GVL_XTS.XtsTransport.GroupItf                   :=   GVL_XTS.CaGroupItf;
GVL_XTS.XtsTransport.GroupInfo                  REF= GVL_XTS.CaGroupInfo;
                                        
GVL_XTS.XtsTransport.MoverItf                   REF= GVL_XTS.MoverItf;
GVL_XTS.XtsTransport.MoverInfo                  REF= GVL_XTS.MoverInfo;
GVL_XTS.XtsTransport.MoverLastPosition          REF= GVL_XTS.LastPosition;
GVL_XTS.XtsTransport.MoverLastGap               REF= GVL_XTS.LastGap;

GVL_XTS.XtsTransport.StationStartIndex          :=   GVL_XTS.StationStartIndex;                                        
GVL_XTS.XtsTransport.StationStart               REF= GVL_XTS.StationStart;      // start position for E_XTS_TRANSPORT_CTRL.CMD_TRANSPORT_START
GVL_XTS.XtsTransport.StationCtrlItf             REF= GVL_XTS.StationCtrlItf;    // station interfaces are required for accessing station methods
GVL_XTS.XtsTransport.StationListsItf            REF= GVL_XTS.StationListItf;    // list interface is required for access to linked list methods
GVL_XTS.XtsTransport.StationControl             REF= GVL_XTS.StationCtrl;
GVL_XTS.XtsTransport.StationState               REF= GVL_XTS.StationState;
//############################################################################
// 	XTS Transport Unit/
//############################################################################
//############################################################################
//############################################################################
// 	/XTS Stations
//############################################################################	
FOR nStation := 1 TO MAX_STATION
DO
  // epimetheus assembles the body
  GVL_XTS.StationListItf[nStation]              := GVL_XTS.StationList[nStation];   // interfaces for list methods
  GVL_XTS.StationCtrlItf[nStation]              := GVL_XTS.Station[nStation];       // interfaces for station methods

  CASE GVL_XTS.StationParameter[nStation].eType
  OF
    //-----------------------------------------------------------------------------
    E_STATION_TYPE.STATION_PROCESS:
      GVL_XTS.Station[nStation].MessageLevel    := GVL_MSG_XTS.MessageLevelStations[nStation];

      GVL_XTS.Station[nStation].StationId       := nStation;  // Know Thyself!

    
      GVL_XTS.Station[nStation].Ctrl            REF= GVL_XTS.StationCtrl;           // station ctrl from extern
      GVL_XTS.Station[nStation].State           REF= GVL_XTS.StationState;          // station state to extern
    
      GVL_XTS.Station[nStation].ItfStations     REF= GVL_XTS.StationListItf;        // give every station all list interfaces for writing mover tickets
      GVL_XTS.Station[nStation].ItfMover        REF= GVL_XTS.MoverItf;              // give every station all mover interfaces for movement in / out of station
      GVL_XTS.Station[nStation].Mover           REF= GVL_XTS.AxisRefMover;          // AXIS_REF to read infos from
      GVL_XTS.Station[nStation].MoverOffset     REF= GVL_XTS.PositionOffset;        // static offsets for all stations, all movers, all stop positions
    
      GVL_XTS.Station[nStation].StationParameter  REF= GVL_XTS.StationParameter;// give every station all station parameters for sending to WaitPos of target station
    
      // cyclic call
      GVL_XTS.Station[nStation].Cycle();                                        // cycle for handshaking with extern
    
      // Queue data for each station
      GVL_XTS.StationQueue[nStation]            := GVL_XTS.StationListItf[nStation].Data;


    //-----------------------------------------------------------------------------
    E_STATION_TYPE.STATION_GEAR_IN_POS:
      GVL_XTS.StationGearIn[nStation].MessageLevel:= GVL_MSG_XTS.MessageLevelStations[nStation];

      GVL_XTS.StationGearIn[nStation].StationId   := nStation;  // Know Thyself!
    
      GVL_XTS.StationGearIn[nStation].Ctrl        REF= GVL_XTS.StationCtrl;           // station ctrl from extern
      GVL_XTS.StationGearIn[nStation].State       REF= GVL_XTS.StationState;          // station state to extern
    
      GVL_XTS.StationGearIn[nStation].ItfStations REF= GVL_XTS.StationListItf;        // give every station all list interfaces for writing mover tickets
      GVL_XTS.StationGearIn[nStation].ItfMover    REF= GVL_XTS.MoverItf;              // give every station all mover interfaces for movement in / out of station
      GVL_XTS.StationGearIn[nStation].Mover       REF= GVL_XTS.AxisRefMover;          // AXIS_REF to read infos from
      GVL_XTS.StationGearIn[nStation].MoverOffset REF= GVL_XTS.PositionOffset;        // static offsets for all stations, all movers, all stop positions
    
    
      GVL_XTS.StationGearIn[nStation].StationParameter  REF= GVL_XTS.StationParameter;// give every station all station parameters for sending to WaitPos of target station
    
      // cyclic call
      GVL_XTS.StationGearIn[nStation].Cycle();                                        // cycle for handshaking with extern
    
      // Queue data for each station
      GVL_XTS.StationQueue[nStation]            := GVL_XTS.StationListItf[nStation].Data;
  ELSE
      //---------------------------------------------------------------------------------
      // no valid station type --> no identity
      //---------------------------------------------------------------------------------
      GVL_XTS.Station[nStation].StationId       := 0; // I am no one
      //---------------------------------------------------------------------------------
  END_CASE
END_FOR
//############################################################################
// 	XTS Stations/
//############################################################################	
//############################################################################
//############################################################################
// 	/XPU environment
//############################################################################	
GVL_XTS.Xpu.XpuInstance                         :=   1;
GVL_XTS.Xpu.MessageLevel                        :=   GVL_MSG_XTS.MessageLevelXpu;

GVL_XTS.Xpu.Ctrl                                REF= GVL_XTS.XpuCtrl;
GVL_XTS.Xpu.State                               REF= GVL_XTS.XpuState;
GVL_XTS.Xpu.XpuModuleInfoData                   REF= GVL_XTS.XpuModules;

GVL_XTS.Xpu.CaGroupOID                          :=   GVL_XTS.CaGroup.GroupInfo.CaGroupOID;

// cyclic call                                
GVL_XTS.Xpu();                                
GVL_XTS.XpuInfo                                 :=   GVL_XTS.Xpu.XpuInfo;
//############################################################################
// 	XPU environment/
//############################################################################	
//############################################################################
//############################################################################	
// 	/CA-Group Class
//############################################################################
// message device identifier
GVL_XTS.CaGroup.MessageDeviceIndex              :=   e_Device.CaGroup + 1;	
// assignment
GVL_XTS.CaGroup.AxisRef                         REF= GVL_XTS.AxisRefMover;
// Interface to Mover methods
GVL_XTS.CaGroup.MoverItf                        REF= GVL_XTS.MoverItf; 
GVL_XTS.CaGroup.GroupRef                        REF= GVL_XTS.CaGroupRef;
GVL_XTS.CaGroup.XpuInfo                         REF= GVL_XTS.XpuInfo;
// cyclic call
GVL_XTS.CaGroup.InfoCycle(TRUE);                // read group status
// InfoData from group
GVL_XTS.CaGroupInfo                             :=   GVL_XTS.CaGroup.GroupInfo;
// Interface of CaGroup
GVL_XTS.CaGroupItf                              :=   GVL_XTS.CaGroup;
//############################################################################	
// 	CA-Group Class/
//############################################################################
//############################################################################
//############################################################################
//  /Mover Class	
//############################################################################	
FOR nMover := 1 TO MAX_MOVER
DO
  GVL_XTS.Mover[nMover].MoverId                 :=   nMover;
  GVL_XTS.Mover[nMover].RailLength              :=   GVL_XTS.Xpu.RailLength;  // mover needs RailLength, in order to calc absolute position from modulo input
  GVL_XTS.Mover[nMover].MessageLevel            :=   GVL_MSG_XTS.MessageLevelMovers[nMover];

  GVL_XTS.Mover[nMover].Ctrl                    REF= GVL_XTS.MoverCtrl;       // mover control from extern
  GVL_XTS.Mover[nMover].State                   REF= GVL_XTS.MoverState;      // mover state to extern

  GVL_XTS.Mover[nMover].MoveData                REF= GVL_XTS.MoveData;        // dyn constraints for extern to write
  GVL_XTS.Mover[nMover].GearData                REF= GVL_XTS.GearData;        // GearIn/GearInPosCa data fro extern to write

  // assignment
  GVL_XTS.Mover[nMover].Mover                   REF= GVL_XTS.AxisRefMover[nMover];  // axis reference to Mover function block
  GVL_XTS.Mover[nMover].LastGap                 REF= GVL_XTS.LastGap[nMover];       // reference to last used gap value datafield
  GVL_XTS.Mover[nMover].LastPosition            REF= GVL_XTS.LastPosition[nMover];  // reference to last position datafield

  GVL_XTS.Mover[nMover].MoverInfo		            REF= GVL_XTS.MoverInfo[nMover];     // refernence to mover info data (ActPos, SetPos, ...)

  GVL_XTS.MoverItf[nMover]                      :=   GVL_XTS.Mover[nMover];

  // cyclic call
  GVL_XTS.Mover[nMover].Cycle();                // call AXIS_REF()
  GVL_XTS.Mover[nMover]();                      // call Ctrl/State
END_FOR
//############################################################################
//  Mover Class/	
//############################################################################	
//############################################################################
//############################################################################
//  /Mover Selector	
//############################################################################
GVL_XTS.MoverSelector.Ctrl                      REF= GVL_XTS.MoverSelectorCtrl;
GVL_XTS.MoverSelector.State                     REF= GVL_XTS.MoverSelectorState;
GVL_XTS.MoverSelector.AxisRef                   REF= GVL_XTS.AxisRefMover;
GVL_XTS.MoverSelector.Info                      REF= GVL_XTS.MoverInfo;
GVL_XTS.MoverSelector.ItfMover                  REF= GVL_XTS.MoverItf;

GVL_XTS.MoverSelector();
//############################################################################
//  Mover Selector/	
//############################################################################	
//############################################################################
//############################################################################
//  /logging
//    - all life is problem solving
//############################################################################
GVL_MSG_XTS.TransportMessageData.Ctrl               REF= GVL_MSG_XTS.TransportMessageCtrl;
GVL_MSG_XTS.TransportMessageData.State              REF= GVL_MSG_XTS.TransportMessageState;
GVL_MSG_XTS.TransportMessageData.MessageIndex       REF= GVL_MSG_XTS.MessageTransportIndex;
GVL_MSG_XTS.TransportMessageData.ErrorIndex         REF= GVL_MSG_XTS.MessageTransportError;
GVL_MSG_XTS.TransportMessageData.DirRoot            :=   ADR(GVL_MSG_XTS.LOG_DIR);
GVL_MSG_XTS.TransportMessageData.FileRoot           :=   ADR(GVL_MSG_XTS.LOG_FILE);
GVL_MSG_XTS.TransportMessageData.MsgList            :=   ADR(GVL_MSG_XTS.TransportMessages);
GVL_MSG_XTS.TransportMessageData.LocalTime          :=   ADR(GVL_MSG_XTS.dtLocalTime);
GVL_MSG_XTS.TransportMessageData();
eMsgState                                       :=   f_GetState   (GVL_MSG_XTS.TransportMessageState.State);
eMsgProgress                                    :=   f_GetProgress(GVL_MSG_XTS.TransportMessageState.State);

CASE eMsgState
OF
  E_MESSAGE_STATE.MSG_STATE_NULL:
    CASE eMsgProgress
    OF
      E_PROGRESS.PROGRESS_INVALID,
      E_PROGRESS.PROGRESS_DONE:
        IF (GVL_MSG_XTS.MessageTransportIndex > GVL_MSG_XTS.MAX_MESSAGE/100) OR
           (GVL_MSG_XTS.MessageTransportError > 0)
        THEN
          GVL_MSG_XTS.TransportMessageCtrl.Cmd      := E_MESSAGE_CTRL.MSG_CTRL_WRITE;
        ELSE
          tonIdleWriteMotion(IN := TRUE, PT:= tIdleWriteMotion);
          IF (tonIdleWriteMotion.Q)
          THEN
            GVL_MSG_XTS.TransportMessageCtrl.Cmd    := E_MESSAGE_CTRL.MSG_CTRL_WRITE;
          END_IF
        END_IF
    END_CASE

  E_MESSAGE_STATE.MSG_STATE_WRITE:
    CASE eMsgProgress
    OF
      E_PROGRESS.PROGRESS_ERROR,
      E_PROGRESS.PROGRESS_DONE:
          tonIdleWriteMotion(IN := FALSE, PT:= tIdleWriteMotion);
        GVL_MSG_XTS.TransportMessageCtrl.Cmd        := E_MESSAGE_CTRL.MSG_CTRL_NULL;
    END_CASE

ELSE
    CASE eMsgProgress
    OF
      E_PROGRESS.PROGRESS_DONE:
        GVL_MSG_XTS.TransportMessageCtrl.Cmd        := E_MESSAGE_CTRL.MSG_CTRL_NULL;
    END_CASE
END_CASE
//############################################################################
//  logging/
//############################################################################
//############################################################################
//############################################################################
//  /Transport Metrics
//############################################################################
GVL_MSG_XTS.MetricsMessageData.Ctrl                 REF= GVL_MSG_XTS.MetricsMessageCtrl;
GVL_MSG_XTS.MetricsMessageData.State                REF= GVL_MSG_XTS.MetricsMessageState;

GVL_MSG_XTS.MetricsMessageData.MessageIndex         REF= GVL_MSG_XTS.MessageMetricsIndex;
GVL_MSG_XTS.MetricsMessageData.ErrorIndex           REF= GVL_MSG_XTS.MessageMetricsError;

GVL_MSG_XTS.MetricsMessageData.DirRoot              :=   ADR(GVL_MSG_XTS.LOG_DIR);
GVL_MSG_XTS.MetricsMessageData.FileRoot             :=   ADR(GVL_MSG_XTS.LOG_FILE_METRIC);

GVL_MSG_XTS.MetricsMessageData.MsgList              :=   ADR(GVL_MSG_XTS.MetricsMessages);
GVL_MSG_XTS.MetricsMessageData.LocalTime            :=   ADR(GVL_MSG_XTS.dtLocalTime);

GVL_MSG_XTS.MetricsMessageData();

eMtrState                                       := f_GetState   (GVL_MSG_XTS.MetricsMessageState.State);
eMtrProgress                                    := f_GetProgress(GVL_MSG_XTS.MetricsMessageState.State);

CASE eMtrState
OF
  E_MESSAGE_STATE.MSG_STATE_NULL:
    CASE eMtrProgress
    OF
      E_PROGRESS.PROGRESS_INVALID:
        IF (GVL_MSG_XTS.MessageMetricsIndex > GVL_MSG_XTS.MAX_MESSAGE/100) OR
           (GVL_MSG_XTS.MessageMetricsError > 0)
        THEN
          GVL_MSG_XTS.MetricsMessageCtrl.Cmd        := E_MESSAGE_CTRL.MSG_CTRL_WRITE;
        ELSE
          tonIdleWriteMetric(IN := TRUE, PT:= tIdleWriteMetric);
          IF (tonIdleWriteMetric.Q)
          THEN
            GVL_MSG_XTS.MetricsMessageCtrl.Cmd      := E_MESSAGE_CTRL.MSG_CTRL_WRITE;
          END_IF
        END_IF
    END_CASE

  E_MESSAGE_STATE.MSG_STATE_WRITE:
    CASE eMtrProgress
    OF
      E_PROGRESS.PROGRESS_ERROR,
      E_PROGRESS.PROGRESS_DONE:
        tonIdleWriteMetric(IN := FALSE, PT:= tIdleWriteMetric);
        GVL_MSG_XTS.MetricsMessageCtrl.Cmd          := E_MESSAGE_CTRL.MSG_CTRL_NULL;
    END_CASE
ELSE
    CASE eMtrProgress
    OF
      E_PROGRESS.PROGRESS_DONE:
        GVL_MSG_XTS.MetricsMessageCtrl.Cmd          := E_MESSAGE_CTRL.MSG_CTRL_NULL;
    END_CASE
END_CASE
//############################################################################
//  Transport Metrics/
//############################################################################
//############################################################################
//############################################################################
//  /Visualization data	
//############################################################################
VisualizationData();
//############################################################################
//  Visualization data/	
//############################################################################

ACTION DefaultStationParameters:
//---------------------------------------------------------------------------------------
//---------------------------------------------------------------------------------------
//
//  Default Station dynamics 
//  - we do not want an array full of nothing 
//  - better have something
//  - leave this initialisation as it is, 
//  - go to MAIN_APP to configure the global datafields
//
//---------------------------------------------------------------------------------------
//---------------------------------------------------------------------------------------
FOR nStn := 1 TO MAX_STATION
DO
  GVL_XTS.StationParameter[nStn].eType               :=   E_STATION_TYPE.INVALID; // make it valid in your configuration
  GVL_XTS.StationParameter[nStn].sText               :=   concat('DEaF_STATION_', TO_STRING(nStn));

  GVL_XTS.StationParameter[nStn].rPosWait            :=   TO_REAL(ABS(GVL_XTS.XpuInfo.rRailLength - nStn*10.0));
  GVL_XTS.StationParameter[nStn].rGap                :=   rInitGap;
  GVL_XTS.StationParameter[nStn].rVelo               :=   rInitVelo;
  GVL_XTS.StationParameter[nStn].rAccDec             :=   rInitAcc;
  GVL_XTS.StationParameter[nStn].rJerk               :=   rInitJerk;
END_FOR
//---------------------------------------------------------------------------------------
//---------------------------------------------------------------------------------------
END_ACTION

ACTION VisualizationData:
//############################################################################
//############################################################################
// Visualization data	
//############################################################################
// get enumerations from XPU for visu:	
eTransportState                       := f_GetState   (GVL_XTS.XtsTransportState.State);
eTransportResult                      := f_GetProgress(GVL_XTS.XtsTransportState.State);

eXpuState                             := f_GetState   (GVL_XTS.XtsTransportState.XpuState.State);
eXpuResult                            := f_GetProgress(GVL_XTS.XtsTransportState.XpuState.State);

eXpuCheck                             := GVL_XTS.XtsTransportState.XpuState.Check;

// display xpu state and result in visu
// get strings and info
sCaGroupState                         := TO_STRING(GVL_XTS.XtsTransportState.GroupInfo.CaGroupState);

sTransportState                       := TO_STRING(eTransportState);
sTransportCheck                       := TO_STRING(GVL_XTS.XtsTransportState.Check);
sTransportResult                      := TO_STRING(eTransportResult);

stXpuStrings.sXpuState                := TO_STRING(eXpuState);
stXpuStrings.sXpuResult               := TO_STRING(eXpuResult);
stXpuStrings.sXpuCyclicCheck          := TO_STRING(eXpuCheck);

stXpuStrings.sXpuOpMode               := GVL_XTS.Xpu.OpModeToString();
stXpuStrings.sXpuMoverId_DetectionMode:= GVL_XTS.Xpu.IdDetectionModeToString();
stXpuStrings.sXpuMoverPosAssignement  := GVL_XTS.Xpu.MoverPositionAssignementToString();

nMoverSelected                        := SEL((nMoverSelected<1), nMoverSelected, 1);
nMoverSelected                        := SEL((nMoverSelected>MAX_MOVER), nMoverSelected, MAX_MOVER);

nStationSelected                      := SEL((nStationSelected<1), nStationSelected, 1);
nStationSelected                      := SEL((nStationSelected>MAX_STATION), nStationSelected, MAX_STATION);

bStationEnable                        := SEL((GVL_XTS.StationCtrl[nStationSelected].Cmd = E_STATION_CTRL.STATION_ENABLE),        FALSE, TRUE);
bStationEnter                         := SEL((GVL_XTS.StationCtrl[nStationSelected].Cmd = E_STATION_CTRL.STATION_MOVER_ENTER),   FALSE, TRUE);
bStationStart                         := SEL((GVL_XTS.StationCtrl[nStationSelected].Cmd = E_STATION_CTRL.STATION_PROCESS_START), FALSE, TRUE);
bStationDone                          := SEL((GVL_XTS.StationCtrl[nStationSelected].Cmd = E_STATION_CTRL.STATION_PROCESS_DONE),  FALSE, TRUE);
bStationOut                           := SEL((GVL_XTS.StationCtrl[nStationSelected].Cmd = E_STATION_CTRL.STATION_MOVER_OUT),     FALSE, TRUE);
bStationGone                          := SEL((GVL_XTS.StationCtrl[nStationSelected].Cmd = E_STATION_CTRL.STATION_MOVER_GONE),    FALSE, TRUE);

eMoverState                           := f_GetState   (GVL_XTS.MoverState[nMoverSelected].State);
eMoverResult                          := f_GetProgress(GVL_XTS.MoverState[nMoverSelected].State);

sMoverState                           := TO_STRING(eMoverState);
sMoverResult                          := TO_STRING(eMoverResult);

eSelectorState                        := f_GetState   (GVL_XTS.MoverSelectorState.State.State);
eSelectorResult                       := f_GetProgress(GVL_XTS.MoverSelectorState.State.State);

sSelectorState                        := TO_STRING(eSelectorState);
sSelectorResult                       := TO_STRING(eSelectorResult);

sStationState                         := TO_STRING(GVL_XTS.StationState[nStationSelected].State);
sStationStateMask                     := Tc2_Utilities.BYTE_TO_BINSTR(GVL_XTS.StationState[nStationSelected].nMask, 8);
sStationCtrlMask                      := Tc2_Utilities.BYTE_TO_BINSTR(GVL_XTS.StationCtrl[nStationSelected].nMask, 8);

tStationSelectedQueue                 := GVL_XTS.StationQueue[nStationSelected];
//############################################################################
//############################################################################
END_ACTION

END_PROGRAM

// ---- APPLICATION/MAIN_APP.TcPOU
//---------------------------------------------------------------------------------------------------------------
//
//  HAUD 2026.03.21
//
//  - MAIN_APPLICATION helper
//    - example PRG for setting up your application startup
//
//---------------------------------------------------------------------------------------------------------------
// This SOFTWARE is provided as an Example by THE PROVIDER "as is" and "with all faults." THE PROVIDER makes no 
// representations or warranties of any kind concerning the safety, suitability, lack of viruses, inaccuracies, 
// typographical errors, or other harmful components of this SOFTWARE. There are inherent dangers in the use of 
// any software, and you are solely responsible for determining whether this SOFTWARE is compatible with your 
// equipment and other software installed on your equipment. You are also solely responsible for the protection 
// of your equipment and backup of your data, and THE PROVIDER will not be liable for any damages you may suffer 
// in connection with using, modifying, or distributing this SOFTWARE.
//---------------------------------------------------------------------------------------------------------------
PROGRAM MAIN_APP
VAR
  eInit      AT %Q*     : E_PROGRESS;   // startup state machine after MAIN is initialized
  bXmlStartup           : BOOL;         // optional example switch for using xml configuration

  rDefaultJerk          : REAL := 400_000.0;
  rDefaultAccDec        : REAL :=  12_500.0;
  rDefaultVeloMax       : REAL :=   3_000.0;
  rDefaultVeloMin       : REAL :=   1_500.0;
  rDefaultGap           : REAL :=      76.0;
END_VAR

//-----------------------------------------------------------------------------
// wait for initialization to be complete before work may start
//-----------------------------------------------------------------------------
IF NOT (MAIN_XTS.eInit = E_PROGRESS.PROGRESS_DONE)
THEN
  eInit                                       := E_PROGRESS.PROGRESS_INIT;
  RETURN;
END_IF
//-----------------------------------------------------------------------------
//-----------------------------------------------------------------------------
// start your application init from here (example)
//-----------------------------------------------------------------------------
CASE eInit
OF
  //---------------------------------------------------------------------------
  E_PROGRESS.PROGRESS_NOT_EXIST:
    RETURN;       // you just bypassed the mapping
                  // check if you require anything from the initialisation
  //---------------------------------------------------------------------------
  E_PROGRESS.PROGRESS_INIT:
    GVL_APPLICATION.ConfigCtrl.Cmd            := E_DATA_CTRL.NULL;
    eInit                                     := E_PROGRESS.PROGRESS_BUSY;

  //---------------------------------------------------------------------------
  E_PROGRESS.PROGRESS_BUSY:
    IF NOT bXmlStartup
    THEN
      StationParameterExample();
      eInit                                   := E_PROGRESS.PROGRESS_WORKING;
    ELSE
      GVL_APPLICATION.ConfigCtrl.Cmd          := E_DATA_CTRL.INIT;
      eInit                                   := E_PROGRESS.PROGRESS_PREPARE;
    END_IF

  //---------------------------------------------------------------------------
  E_PROGRESS.PROGRESS_PREPARE:
    IF (GVL_APPLICATION.ConfigState.State = E_DATA_STATE.INIT + E_PROGRESS.PROGRESS_DONE)
    THEN
      GVL_APPLICATION.ConfigCtrl.Cmd          := E_DATA_CTRL.READ;
      eInit                                   := E_PROGRESS.PROGRESS_STARTUP;
    END_IF

  E_PROGRESS.PROGRESS_STARTUP:
    IF (GVL_APPLICATION.ConfigState.State = E_DATA_STATE.READ + E_PROGRESS.PROGRESS_DONE)
    THEN
      GVL_APPLICATION.ConfigCtrl.Cmd          := E_DATA_CTRL.NULL;
      eInit                                   := E_PROGRESS.PROGRESS_CHECK;
    END_IF

  E_PROGRESS.PROGRESS_CHECK:
    eInit                                     := E_PROGRESS.PROGRESS_OCCUPIED;

  E_PROGRESS.PROGRESS_OCCUPIED:
    eInit                                     := E_PROGRESS.PROGRESS_WORKING;

  E_PROGRESS.PROGRESS_WORKING:
    eInit                                     := E_PROGRESS.PROGRESS_DONE;
END_CASE
//-----------------------------------------------------------------------------
//-----------------------------------------------------------------------------
//-----------------------------------------------------------------------------
// connect data and control to xml configuration
GVL_APPLICATION.StationConfig.Identity        :=   GVL_XTS.Xpu.XpuOtcid;
GVL_APPLICATION.StationConfig.Ctrl            REF= GVL_APPLICATION.ConfigCtrl;
GVL_APPLICATION.StationConfig.State           REF= GVL_APPLICATION.ConfigState;

GVL_APPLICATION.StationConfig.MessageDevice   := e_Device.Device_Configuration;
GVL_APPLICATION.StationConfig.MessageLevel    := GVL_MSG_XTS.MessageLevel;
GVL_APPLICATION.StationConfig.FolderPath      := GVL_MSG_XTS.CON_DIR;
GVL_APPLICATION.StationConfig.StationParameter:= ADR(GVL_XTS.StationParameter);

GVL_APPLICATION.StationConfig();        // call xml configuration
//-----------------------------------------------------------------------------
//-----------------------------------------------------------------------------

END_PROGRAM

// ---- APPLICATION/StationParameterExample.TcPOU
FUNCTION StationParameterExample  : BOOL
VAR
  nStationParameter                 : UINT; // THIS IS ONLY FOR EXAMPLE USE, CHECK MAX_STATION MANUALLY
END_VAR

//-----------------------------------------------------------------------------------------------------------------------------------------
//-----------------------------------------------------------------------------------------------------------------------------------------
//
//  HAUD 2026.06.01
//
//  - hard coded station parameters as example
//  - TODO: xml DataServer implementation for station parameter read/write
//
//  - reminder: (this you HAVE to check manually when setting up the transport)
//-----------------------------------------------------------------------------
//    - DO NOT place the modulo turn within the range of a station
//
//    - in case the extern process requires multiple xts stations, 
//      - the range must be closed and in strict order
//-----------------------------------------------------------------------------------------------------------------------------------------
//-----------------------------------------------------------------------------------------------------------------------------------------
GVL_XTS.StationStartIndex                                         := 150;
GVL_XTS.StationStart.rPosWait                                     :=   1900.0; // for every TRANSPORT_START this physical position may differ from the rPosWait of StationStartIndex station

GVL_XTS.StationStart.rGap                                         :=     78.0;
GVL_XTS.StationStart.rVelo                                        :=   1500.0;
GVL_XTS.StationStart.rAccDec                                      :=  12500.0;
GVL_XTS.StationStart.rJerk                                        := 400000.0;

FOR nStationParameter := 1 TO GVL_XTS_CONSTANTS.MAX_STATION
DO
  GVL_XTS.StationParameter[nStationParameter].eType               := E_STATION_TYPE.STATION_PROCESS;
  GVL_XTS.StationParameter[nStationParameter].rGap                := MAIN_APP.rDefaultGap;
  GVL_XTS.StationParameter[nStationParameter].rVelo               := MAIN_APP.rDefaultVeloMax;
  GVL_XTS.StationParameter[nStationParameter].rAccDec             := MAIN_APP.rDefaultAccDec;
  GVL_XTS.StationParameter[nStationParameter].rJerk               := MAIN_APP.rDefaultJerk;
END_FOR
//-----------------------------------------------------------------------------------------------------------------------------------------
//  PRC 01
//-----------------------------------------------------------------------------------------------------------------------------------------
FOR nStationParameter := 1 TO 16
DO
  GVL_XTS.StationParameter[nStationParameter].rVelo               := MAIN_APP.rDefaultVeloMin;
END_FOR
nStationParameter := 1;
GVL_XTS.StationParameter[nStationParameter].eType                 := E_STATION_TYPE.STATION_PROCESS;
GVL_XTS.StationParameter[nStationParameter].sText                 := 'PRC_01_01';
GVL_XTS.StationParameter[nStationParameter].nConfiguredStopCount  :=       1;   // how many stops the mover has to make in this station

GVL_XTS.StationParameter[nStationParameter].rPosWait              :=    2000.0; // absolute modulo position
GVL_XTS.StationParameter[nStationParameter].rPosStop[1]           :=      80.0; // relative to rPosWait
GVL_XTS.StationParameter[nStationParameter].rReleaseDistance      :=    1280.0; // relative to Mover.ActPos

nStationParameter := 2;
GVL_XTS.StationParameter[nStationParameter].eType                 := E_STATION_TYPE.STATION_PROCESS;
GVL_XTS.StationParameter[nStationParameter].sText                 := 'PRC_01_02';
GVL_XTS.StationParameter[nStationParameter].nConfiguredStopCount  :=       1;   // how many stops the mover has to make in this station

GVL_XTS.StationParameter[nStationParameter].rPosWait              :=    2000.0; // absolute modulo position
GVL_XTS.StationParameter[nStationParameter].rPosStop[1]           :=     160.0; // relative to rPosWait
GVL_XTS.StationParameter[nStationParameter].rReleaseDistance      :=    1200.0; // relative to Mover.ActPos

nStationParameter := 3;
GVL_XTS.StationParameter[nStationParameter].eType                 := E_STATION_TYPE.STATION_PROCESS;
GVL_XTS.StationParameter[nStationParameter].sText                 := 'PRC_01_03';
GVL_XTS.StationParameter[nStationParameter].nConfiguredStopCount  :=       1;   // how many stops the mover has to make in this station

GVL_XTS.StationParameter[nStationParameter].rPosWait              :=    2000.0; // absolute modulo position
GVL_XTS.StationParameter[nStationParameter].rPosStop[1]           :=     240.0; // relative to rPosWait
GVL_XTS.StationParameter[nStationParameter].rReleaseDistance      :=    1120.0; // relative to Mover.ActPos

nStationParameter := 4;
GVL_XTS.StationParameter[nStationParameter].eType                 := E_STATION_TYPE.STATION_PROCESS;
GVL_XTS.StationParameter[nStationParameter].sText                 := 'PRC_01_04';
GVL_XTS.StationParameter[nStationParameter].nConfiguredStopCount  :=       1;   // how many stops the mover has to make in this station

GVL_XTS.StationParameter[nStationParameter].rPosWait              :=    2000.0; // absolute modulo position
GVL_XTS.StationParameter[nStationParameter].rPosStop[1]           :=     320.0; // relative to rPosWait
GVL_XTS.StationParameter[nStationParameter].rReleaseDistance      :=    1040.0; // relative to Mover.ActPos

nStationParameter := 5;
GVL_XTS.StationParameter[nStationParameter].eType                 := E_STATION_TYPE.STATION_PROCESS;
GVL_XTS.StationParameter[nStationParameter].sText                 := 'PRC_01_05';
GVL_XTS.StationParameter[nStationParameter].nConfiguredStopCount  :=       1;   // how many stops the mover has to make in this station

GVL_XTS.StationParameter[nStationParameter].rPosWait              :=    2000.0; // absolute modulo position
GVL_XTS.StationParameter[nStationParameter].rPosStop[1]           :=     400.0; // relative to rPosWait
GVL_XTS.StationParameter[nStationParameter].rReleaseDistance      :=     960.0; // relative to Mover.ActPos

nStationParameter := 6;
GVL_XTS.StationParameter[nStationParameter].eType                 := E_STATION_TYPE.STATION_PROCESS;
GVL_XTS.StationParameter[nStationParameter].sText                 := 'PRC_01_06';
GVL_XTS.StationParameter[nStationParameter].nConfiguredStopCount  :=       1;   // how many stops the mover has to make in this station

GVL_XTS.StationParameter[nStationParameter].rPosWait              :=    2000.0; // absolute modulo position
GVL_XTS.StationParameter[nStationParameter].rPosStop[1]           :=     480.0; // relative to rPosWait
GVL_XTS.StationParameter[nStationParameter].rReleaseDistance      :=     880.0; // relative to Mover.ActPos

nStationParameter := 7;
GVL_XTS.StationParameter[nStationParameter].eType                 := E_STATION_TYPE.STATION_PROCESS;
GVL_XTS.StationParameter[nStationParameter].sText                 := 'PRC_01_07';
GVL_XTS.StationParameter[nStationParameter].nConfiguredStopCount  :=       1;   // how many stops the mover has to make in this station

GVL_XTS.StationParameter[nStationParameter].rPosWait              :=    2000.0; // absolute modulo position
GVL_XTS.StationParameter[nStationParameter].rPosStop[1]           :=     560.0; // relative to rPosWait
GVL_XTS.StationParameter[nStationParameter].rReleaseDistance      :=     800.0; // relative to Mover.ActPos

nStationParameter := 8;
GVL_XTS.StationParameter[nStationParameter].eType                 := E_STATION_TYPE.STATION_PROCESS;
GVL_XTS.StationParameter[nStationParameter].sText                 := 'PRC_01_08';
GVL_XTS.StationParameter[nStationParameter].nConfiguredStopCount  :=       1;   // how many stops the mover has to make in this station

GVL_XTS.StationParameter[nStationParameter].rPosWait              :=    2000.0; // absolute modulo position
GVL_XTS.StationParameter[nStationParameter].rPosStop[1]           :=     640.0; // relative to rPosWait
GVL_XTS.StationParameter[nStationParameter].rReleaseDistance      :=     720.0; // relative to Mover.ActPos

nStationParameter := 9;
GVL_XTS.StationParameter[nStationParameter].eType                 := E_STATION_TYPE.STATION_PROCESS;
GVL_XTS.StationParameter[nStationParameter].sText                 := 'PRC_01_09';
GVL_XTS.StationParameter[nStationParameter].nConfiguredStopCount  :=       1;   // how many stops the mover has to make in this station

GVL_XTS.StationParameter[nStationParameter].rPosWait              :=    2000.0; // absolute modulo position
GVL_XTS.StationParameter[nStationParameter].rPosStop[1]           :=     720.0; // relative to rPosWait
GVL_XTS.StationParameter[nStationParameter].rReleaseDistance      :=     640.0; // relative to Mover.ActPos

nStationParameter := 10;
GVL_XTS.StationParameter[nStationParameter].eType                 := E_STATION_TYPE.STATION_PROCESS;
GVL_XTS.StationParameter[nStationParameter].sText                 := 'PRC_01_10';
GVL_XTS.StationParameter[nStationParameter].nConfiguredStopCount  :=       1;   // how many stops the mover has to make in this station

GVL_XTS.StationParameter[nStationParameter].rPosWait              :=    2000.0; // absolute modulo position
GVL_XTS.StationParameter[nStationParameter].rPosStop[1]           :=     800.0; // relative to rPosWait
GVL_XTS.StationParameter[nStationParameter].rReleaseDistance      :=     560.0; // relative to Mover.ActPos

nStationParameter := 11;
GVL_XTS.StationParameter[nStationParameter].eType                 := E_STATION_TYPE.STATION_PROCESS;
GVL_XTS.StationParameter[nStationParameter].sText                 := 'PRC_01_11';
GVL_XTS.StationParameter[nStationParameter].nConfiguredStopCount  :=       1;   // how many stops the mover has to make in this station

GVL_XTS.StationParameter[nStationParameter].rPosWait              :=    2000.0; // absolute modulo position
GVL_XTS.StationParameter[nStationParameter].rPosStop[1]           :=     880.0; // relative to rPosWait
GVL_XTS.StationParameter[nStationParameter].rReleaseDistance      :=     480.0; // relative to Mover.ActPos

nStationParameter := 12;
GVL_XTS.StationParameter[nStationParameter].eType                 := E_STATION_TYPE.STATION_PROCESS;
GVL_XTS.StationParameter[nStationParameter].sText                 := 'PRC_01_12';
GVL_XTS.StationParameter[nStationParameter].nConfiguredStopCount  :=       1;   // how many stops the mover has to make in this station

GVL_XTS.StationParameter[nStationParameter].rPosWait              :=    2000.0; // absolute modulo position
GVL_XTS.StationParameter[nStationParameter].rPosStop[1]           :=     960.0; // relative to rPosWait
GVL_XTS.StationParameter[nStationParameter].rReleaseDistance      :=     400.0; // relative to Mover.ActPos

nStationParameter := 13;
GVL_XTS.StationParameter[nStationParameter].eType                 := E_STATION_TYPE.STATION_PROCESS;
GVL_XTS.StationParameter[nStationParameter].sText                 := 'PRC_01_13';
GVL_XTS.StationParameter[nStationParameter].nConfiguredStopCount  :=       1;   // how many stops the mover has to make in this station

GVL_XTS.StationParameter[nStationParameter].rPosWait              :=    2000.0; // absolute modulo position
GVL_XTS.StationParameter[nStationParameter].rPosStop[1]           :=    1040.0; // relative to rPosWait
GVL_XTS.StationParameter[nStationParameter].rReleaseDistance      :=     320.0; // relative to Mover.ActPos

nStationParameter := 14;
GVL_XTS.StationParameter[nStationParameter].eType                 := E_STATION_TYPE.STATION_PROCESS;
GVL_XTS.StationParameter[nStationParameter].sText                 := 'PRC_01_14';
GVL_XTS.StationParameter[nStationParameter].nConfiguredStopCount  :=       1;   // how many stops the mover has to make in this station

GVL_XTS.StationParameter[nStationParameter].rPosWait              :=    2000.0; // absolute modulo position
GVL_XTS.StationParameter[nStationParameter].rPosStop[1]           :=    1120.0; // relative to rPosWait
GVL_XTS.StationParameter[nStationParameter].rReleaseDistance      :=     240.0; // relative to Mover.ActPos

nStationParameter := 15;
GVL_XTS.StationParameter[nStationParameter].eType                 := E_STATION_TYPE.STATION_PROCESS;
GVL_XTS.StationParameter[nStationParameter].sText                 := 'PRC_01_15';
GVL_XTS.StationParameter[nStationParameter].nConfiguredStopCount  :=       1;   // how many stops the mover has to make in this station

GVL_XTS.StationParameter[nStationParameter].rPosWait              :=    2000.0; // absolute modulo position
GVL_XTS.StationParameter[nStationParameter].rPosStop[1]           :=    1200.0; // relative to rPosWait
GVL_XTS.StationParameter[nStationParameter].rReleaseDistance      :=     160.0; // relative to Mover.ActPos

nStationParameter := 16;
GVL_XTS.StationParameter[nStationParameter].eType                 := E_STATION_TYPE.STATION_PROCESS;
GVL_XTS.StationParameter[nStationParameter].sText                 := 'PRC_01_16';
GVL_XTS.StationParameter[nStationParameter].nConfiguredStopCount  :=       1;   // how many stops the mover has to make in this station

GVL_XTS.StationParameter[nStationParameter].rPosWait              :=    2000.0; // absolute modulo position
GVL_XTS.StationParameter[nStationParameter].rPosStop[1]           :=    1280.0; // relative to rPosWait
GVL_XTS.StationParameter[nStationParameter].rReleaseDistance      :=      25.0; // relative to Mover.ActPos

//-----------------------------------------------------------------------------------------------------------------------------------------
// PRC 03 
//-----------------------------------------------------------------------------------------------------------------------------------------
nStationParameter := 20;
GVL_XTS.StationParameter[nStationParameter].eType                 := E_STATION_TYPE.STATION_PROCESS;
GVL_XTS.StationParameter[nStationParameter].sText                 := 'PRC_03_01';
GVL_XTS.StationParameter[nStationParameter].nConfiguredStopCount  :=       1;   // how many stops the mover has to make in this station

GVL_XTS.StationParameter[nStationParameter].rPosWait              :=    5000.0; // absolute modulo position
GVL_XTS.StationParameter[nStationParameter].rPosStop[1]           :=      80.0; // relative to rPosWait
GVL_XTS.StationParameter[nStationParameter].rReleaseDistance      :=    1280.0; // relative to Mover.ActPos

nStationParameter := 21;
GVL_XTS.StationParameter[nStationParameter].eType                 := E_STATION_TYPE.STATION_PROCESS;
GVL_XTS.StationParameter[nStationParameter].sText                 := 'PRC_03_02';
GVL_XTS.StationParameter[nStationParameter].nConfiguredStopCount  :=       1;   // how many stops the mover has to make in this station

GVL_XTS.StationParameter[nStationParameter].rPosWait              :=    5000.0; // absolute modulo position
GVL_XTS.StationParameter[nStationParameter].rPosStop[1]           :=     160.0; // relative to rPosWait
GVL_XTS.StationParameter[nStationParameter].rReleaseDistance      :=    1200.0; // relative to Mover.ActPos

nStationParameter := 22;
GVL_XTS.StationParameter[nStationParameter].eType                 := E_STATION_TYPE.STATION_PROCESS;
GVL_XTS.StationParameter[nStationParameter].sText                 := 'PRC_03_03';
GVL_XTS.StationParameter[nStationParameter].nConfiguredStopCount  :=       1;   // how many stops the mover has to make in this station

GVL_XTS.StationParameter[nStationParameter].rPosWait              :=    5000.0; // absolute modulo position
GVL_XTS.StationParameter[nStationParameter].rPosStop[1]           :=     240.0; // relative to rPosWait
GVL_XTS.StationParameter[nStationParameter].rReleaseDistance      :=    1120.0; // relative to Mover.ActPos

nStationParameter := 23;
GVL_XTS.StationParameter[nStationParameter].eType                 := E_STATION_TYPE.STATION_PROCESS;
GVL_XTS.StationParameter[nStationParameter].sText                 := 'PRC_03_04';
GVL_XTS.StationParameter[nStationParameter].nConfiguredStopCount  :=       1;   // how many stops the mover has to make in this station

GVL_XTS.StationParameter[nStationParameter].rPosWait              :=    5000.0; // absolute modulo position
GVL_XTS.StationParameter[nStationParameter].rPosStop[1]           :=     320.0; // relative to rPosWait
GVL_XTS.StationParameter[nStationParameter].rReleaseDistance      :=    1040.0; // relative to Mover.ActPos

nStationParameter := 24;
GVL_XTS.StationParameter[nStationParameter].eType                 := E_STATION_TYPE.STATION_PROCESS;
GVL_XTS.StationParameter[nStationParameter].sText                 := 'PRC_03_05';
GVL_XTS.StationParameter[nStationParameter].nConfiguredStopCount  :=       1;   // how many stops the mover has to make in this station

GVL_XTS.StationParameter[nStationParameter].rPosWait              :=    5000.0; // absolute modulo position
GVL_XTS.StationParameter[nStationParameter].rPosStop[1]           :=     400.0; // relative to rPosWait
GVL_XTS.StationParameter[nStationParameter].rReleaseDistance      :=     960.0; // relative to Mover.ActPos

nStationParameter := 25;
GVL_XTS.StationParameter[nStationParameter].eType                 := E_STATION_TYPE.STATION_PROCESS;
GVL_XTS.StationParameter[nStationParameter].sText                 := 'PRC_03_06';
GVL_XTS.StationParameter[nStationParameter].nConfiguredStopCount  :=       1;   // how many stops the mover has to make in this station

GVL_XTS.StationParameter[nStationParameter].rPosWait              :=    5000.0; // absolute modulo position
GVL_XTS.StationParameter[nStationParameter].rPosStop[1]           :=     480.0; // relative to rPosWait
GVL_XTS.StationParameter[nStationParameter].rReleaseDistance      :=     880.0; // relative to Mover.ActPos

nStationParameter := 26;
GVL_XTS.StationParameter[nStationParameter].eType                 := E_STATION_TYPE.STATION_PROCESS;
GVL_XTS.StationParameter[nStationParameter].sText                 := 'PRC_03_07';
GVL_XTS.StationParameter[nStationParameter].nConfiguredStopCount  :=       1;   // how many stops the mover has to make in this station

GVL_XTS.StationParameter[nStationParameter].rPosWait              :=    5000.0; // absolute modulo position
GVL_XTS.StationParameter[nStationParameter].rPosStop[1]           :=     560.0; // relative to rPosWait
GVL_XTS.StationParameter[nStationParameter].rReleaseDistance      :=     800.0; // relative to Mover.ActPos

nStationParameter := 27;
GVL_XTS.StationParameter[nStationParameter].eType                 := E_STATION_TYPE.STATION_PROCESS;
GVL_XTS.StationParameter[nStationParameter].sText                 := 'PRC_03_08';
GVL_XTS.StationParameter[nStationParameter].nConfiguredStopCount  :=       1;   // how many stops the mover has to make in this station

GVL_XTS.StationParameter[nStationParameter].rPosWait              :=    5000.0; // absolute modulo position
GVL_XTS.StationParameter[nStationParameter].rPosStop[1]           :=     640.0; // relative to rPosWait
GVL_XTS.StationParameter[nStationParameter].rReleaseDistance      :=     720.0; // relative to Mover.ActPos

nStationParameter := 28;
GVL_XTS.StationParameter[nStationParameter].eType                 := E_STATION_TYPE.STATION_PROCESS;
GVL_XTS.StationParameter[nStationParameter].sText                 := 'PRC_03_09';
GVL_XTS.StationParameter[nStationParameter].nConfiguredStopCount  :=       1;   // how many stops the mover has to make in this station

GVL_XTS.StationParameter[nStationParameter].rPosWait              :=    5000.0; // absolute modulo position
GVL_XTS.StationParameter[nStationParameter].rPosStop[1]           :=     720.0; // relative to rPosWait
GVL_XTS.StationParameter[nStationParameter].rReleaseDistance      :=     640.0; // relative to Mover.ActPos

nStationParameter := 29;
GVL_XTS.StationParameter[nStationParameter].eType                 := E_STATION_TYPE.STATION_PROCESS;
GVL_XTS.StationParameter[nStationParameter].sText                 := 'PRC_03_10';
GVL_XTS.StationParameter[nStationParameter].nConfiguredStopCount  :=       1;   // how many stops the mover has to make in this station

GVL_XTS.StationParameter[nStationParameter].rPosWait              :=    5000.0; // absolute modulo position
GVL_XTS.StationParameter[nStationParameter].rPosStop[1]           :=     800.0; // relative to rPosWait
GVL_XTS.StationParameter[nStationParameter].rReleaseDistance      :=     560.0; // relative to Mover.ActPos

nStationParameter := 30;
GVL_XTS.StationParameter[nStationParameter].eType                 := E_STATION_TYPE.STATION_PROCESS;
GVL_XTS.StationParameter[nStationParameter].sText                 := 'PRC_03_11';
GVL_XTS.StationParameter[nStationParameter].nConfiguredStopCount  :=       1;   // how many stops the mover has to make in this station

GVL_XTS.StationParameter[nStationParameter].rPosWait              :=    5000.0; // absolute modulo position
GVL_XTS.StationParameter[nStationParameter].rPosStop[1]           :=     880.0; // relative to rPosWait
GVL_XTS.StationParameter[nStationParameter].rReleaseDistance      :=     480.0; // relative to Mover.ActPos

nStationParameter := 31;
GVL_XTS.StationParameter[nStationParameter].eType                 := E_STATION_TYPE.STATION_PROCESS;
GVL_XTS.StationParameter[nStationParameter].sText                 := 'PRC_03_12';
GVL_XTS.StationParameter[nStationParameter].nConfiguredStopCount  :=       1;   // how many stops the mover has to make in this station

GVL_XTS.StationParameter[nStationParameter].rPosWait              :=    5000.0; // absolute modulo position
GVL_XTS.StationParameter[nStationParameter].rPosStop[1]           :=     960.0; // relative to rPosWait
GVL_XTS.StationParameter[nStationParameter].rReleaseDistance      :=     400.0; // relative to Mover.ActPos

nStationParameter := 32;
GVL_XTS.StationParameter[nStationParameter].eType                 := E_STATION_TYPE.STATION_PROCESS;
GVL_XTS.StationParameter[nStationParameter].sText                 := 'PRC_03_13';
GVL_XTS.StationParameter[nStationParameter].nConfiguredStopCount  :=       1;   // how many stops the mover has to make in this station

GVL_XTS.StationParameter[nStationParameter].rPosWait              :=    5000.0; // absolute modulo position
GVL_XTS.StationParameter[nStationParameter].rPosStop[1]           :=    1040.0; // relative to rPosWait
GVL_XTS.StationParameter[nStationParameter].rReleaseDistance      :=     320.0; // relative to Mover.ActPos

nStationParameter := 33;
GVL_XTS.StationParameter[nStationParameter].eType                 := E_STATION_TYPE.STATION_PROCESS;
GVL_XTS.StationParameter[nStationParameter].sText                 := 'PRC_03_14';
GVL_XTS.StationParameter[nStationParameter].nConfiguredStopCount  :=       1;   // how many stops the mover has to make in this station

GVL_XTS.StationParameter[nStationParameter].rPosWait              :=    5000.0; // absolute modulo position
GVL_XTS.StationParameter[nStationParameter].rPosStop[1]           :=    1120.0; // relative to rPosWait
GVL_XTS.StationParameter[nStationParameter].rReleaseDistance      :=     240.0; // relative to Mover.ActPos

nStationParameter := 34;
GVL_XTS.StationParameter[nStationParameter].eType                 := E_STATION_TYPE.STATION_PROCESS;
GVL_XTS.StationParameter[nStationParameter].sText                 := 'PRC_03_15';
GVL_XTS.StationParameter[nStationParameter].nConfiguredStopCount  :=       1;   // how many stops the mover has to make in this station

GVL_XTS.StationParameter[nStationParameter].rPosWait              :=    5000.0; // absolute modulo position
GVL_XTS.StationParameter[nStationParameter].rPosStop[1]           :=    1200.0; // relative to rPosWait
GVL_XTS.StationParameter[nStationParameter].rReleaseDistance      :=     160.0; // relative to Mover.ActPos

nStationParameter := 35;
GVL_XTS.StationParameter[nStationParameter].eType                 := E_STATION_TYPE.STATION_PROCESS;
GVL_XTS.StationParameter[nStationParameter].sText                 := 'PRC_03_16';
GVL_XTS.StationParameter[nStationParameter].nConfiguredStopCount  :=       1;   // how many stops the mover has to make in this station

GVL_XTS.StationParameter[nStationParameter].rPosWait              :=    5000.0; // absolute modulo position
GVL_XTS.StationParameter[nStationParameter].rPosStop[1]           :=    1280.0; // relative to rPosWait
GVL_XTS.StationParameter[nStationParameter].rReleaseDistance      :=      25.0; // relative to Mover.ActPos

//-----------------------------------------------------------------------------------------------------------------------------------------
// PRC 04 
//-----------------------------------------------------------------------------------------------------------------------------------------
nStationParameter := 37;
GVL_XTS.StationParameter[nStationParameter].eType                 := E_STATION_TYPE.STATION_PROCESS;
GVL_XTS.StationParameter[nStationParameter].sText                 := 'PRC_04';
GVL_XTS.StationParameter[nStationParameter].nConfiguredStopCount  :=       1;   // how many stops the mover has to make in this station

GVL_XTS.StationParameter[nStationParameter].rPosWait              :=    7500.0; // absolute modulo position
GVL_XTS.StationParameter[nStationParameter].rPosStop[1]           :=       0.0; // relative to rPosWait
GVL_XTS.StationParameter[nStationParameter].rReleaseDistance      :=      50.0; // relative to Mover.ActPos
GVL_XTS.StationParameter[nStationParameter].rVelo                 :=     500.0;

//-----------------------------------------------------------------------------------------------------------------------------------------
// PRC 05
//-----------------------------------------------------------------------------------------------------------------------------------------
nStationParameter := 45;
GVL_XTS.StationParameter[nStationParameter].eType                 := E_STATION_TYPE.STATION_PROCESS;
GVL_XTS.StationParameter[nStationParameter].sText                 := 'PRC_05_01';
GVL_XTS.StationParameter[nStationParameter].nConfiguredStopCount  :=       1;   // how many stops the mover has to make in this station

GVL_XTS.StationParameter[nStationParameter].rPosWait              :=    8250.0; // absolute modulo position
GVL_XTS.StationParameter[nStationParameter].rPosStop[1]           :=      80.0; // relative to rPosWait
GVL_XTS.StationParameter[nStationParameter].rReleaseDistance      :=     560.0; // relative to Mover.ActPos

nStationParameter := 46;
GVL_XTS.StationParameter[nStationParameter].eType                 := E_STATION_TYPE.STATION_PROCESS;
GVL_XTS.StationParameter[nStationParameter].sText                 := 'PRC_05_02';
GVL_XTS.StationParameter[nStationParameter].nConfiguredStopCount  :=       1;   // how many stops the mover has to make in this station

GVL_XTS.StationParameter[nStationParameter].rPosWait              :=    8250.0; // absolute modulo position
GVL_XTS.StationParameter[nStationParameter].rPosStop[1]           :=     160.0; // relative to rPosWait
GVL_XTS.StationParameter[nStationParameter].rReleaseDistance      :=     480.0; // relative to Mover.ActPos

nStationParameter := 47;
GVL_XTS.StationParameter[nStationParameter].eType                 := E_STATION_TYPE.STATION_PROCESS;
GVL_XTS.StationParameter[nStationParameter].sText                 := 'PRC_05_03';
GVL_XTS.StationParameter[nStationParameter].nConfiguredStopCount  :=       1;   // how many stops the mover has to make in this station

GVL_XTS.StationParameter[nStationParameter].rPosWait              :=    8250.0; // absolute modulo position
GVL_XTS.StationParameter[nStationParameter].rPosStop[1]           :=     240.0; // relative to rPosWait
GVL_XTS.StationParameter[nStationParameter].rReleaseDistance      :=     400.0; // relative to Mover.ActPos

nStationParameter := 48;
GVL_XTS.StationParameter[nStationParameter].eType                 := E_STATION_TYPE.STATION_PROCESS;
GVL_XTS.StationParameter[nStationParameter].sText                 := 'PRC_05_04';
GVL_XTS.StationParameter[nStationParameter].nConfiguredStopCount  :=       1;   // how many stops the mover has to make in this station

GVL_XTS.StationParameter[nStationParameter].rPosWait              :=    8250.0; // absolute modulo position
GVL_XTS.StationParameter[nStationParameter].rPosStop[1]           :=     320.0; // relative to rPosWait
GVL_XTS.StationParameter[nStationParameter].rReleaseDistance      :=     320.0; // relative to Mover.ActPos

nStationParameter := 49;
GVL_XTS.StationParameter[nStationParameter].eType                 := E_STATION_TYPE.STATION_PROCESS;
GVL_XTS.StationParameter[nStationParameter].sText                 := 'PRC_05_05';
GVL_XTS.StationParameter[nStationParameter].nConfiguredStopCount  :=       1;   // how many stops the mover has to make in this station

GVL_XTS.StationParameter[nStationParameter].rPosWait              :=    8250.0; // absolute modulo position
GVL_XTS.StationParameter[nStationParameter].rPosStop[1]           :=     400.0; // relative to rPosWait
GVL_XTS.StationParameter[nStationParameter].rReleaseDistance      :=     240.0; // relative to Mover.ActPos

nStationParameter := 50;
GVL_XTS.StationParameter[nStationParameter].eType                 := E_STATION_TYPE.STATION_PROCESS;
GVL_XTS.StationParameter[nStationParameter].sText                 := 'PRC_05_06';
GVL_XTS.StationParameter[nStationParameter].nConfiguredStopCount  :=       1;   // how many stops the mover has to make in this station

GVL_XTS.StationParameter[nStationParameter].rPosWait              :=    8250.0; // absolute modulo position
GVL_XTS.StationParameter[nStationParameter].rPosStop[1]           :=     480.0; // relative to rPosWait
GVL_XTS.StationParameter[nStationParameter].rReleaseDistance      :=     160.0; // relative to Mover.ActPos

nStationParameter := 51;
GVL_XTS.StationParameter[nStationParameter].eType                 := E_STATION_TYPE.STATION_PROCESS;
GVL_XTS.StationParameter[nStationParameter].sText                 := 'PRC_05_07';
GVL_XTS.StationParameter[nStationParameter].nConfiguredStopCount  :=       1;   // how many stops the mover has to make in this station

GVL_XTS.StationParameter[nStationParameter].rPosWait              :=    8250.0; // absolute modulo position
GVL_XTS.StationParameter[nStationParameter].rPosStop[1]           :=     560.0; // relative to rPosWait
GVL_XTS.StationParameter[nStationParameter].rReleaseDistance      :=      80.0; // relative to Mover.ActPos

nStationParameter := 52;
GVL_XTS.StationParameter[nStationParameter].eType                 := E_STATION_TYPE.STATION_PROCESS;
GVL_XTS.StationParameter[nStationParameter].sText                 := 'PRC_05_08';
GVL_XTS.StationParameter[nStationParameter].nConfiguredStopCount  :=       1;   // how many stops the mover has to make in this station

GVL_XTS.StationParameter[nStationParameter].rPosWait              :=    8250.0; // absolute modulo position
GVL_XTS.StationParameter[nStationParameter].rPosStop[1]           :=     640.0; // relative to rPosWait
GVL_XTS.StationParameter[nStationParameter].rReleaseDistance      :=      25.0; // relative to Mover.ActPos
//-----------------------------------------------------------------------------------------------------------------------------------------
// PRC 06 
//-----------------------------------------------------------------------------------------------------------------------------------------
FOR nStationParameter := 58 TO 69
DO
  GVL_XTS.StationParameter[nStationParameter].rVelo               := MAIN_APP.rDefaultVeloMin;
END_FOR
nStationParameter := 58;
GVL_XTS.StationParameter[nStationParameter].eType                 := E_STATION_TYPE.STATION_PROCESS;
GVL_XTS.StationParameter[nStationParameter].sText                 := 'PRC_06_01';
GVL_XTS.StationParameter[nStationParameter].nConfiguredStopCount  :=       1;   // how many stops the mover has to make in this station

GVL_XTS.StationParameter[nStationParameter].rPosWait              :=    9500.0; // absolute modulo position
GVL_XTS.StationParameter[nStationParameter].rPosStop[1]           :=      80.0; // relative to rPosWait
GVL_XTS.StationParameter[nStationParameter].rReleaseDistance      :=     880.0; // relative to Mover.ActPos

nStationParameter := 59;
GVL_XTS.StationParameter[nStationParameter].eType                 := E_STATION_TYPE.STATION_PROCESS;
GVL_XTS.StationParameter[nStationParameter].sText                 := 'PRC_06_02';
GVL_XTS.StationParameter[nStationParameter].nConfiguredStopCount  :=       1;   // how many stops the mover has to make in this station

GVL_XTS.StationParameter[nStationParameter].rPosWait              :=    9500.0; // absolute modulo position
GVL_XTS.StationParameter[nStationParameter].rPosStop[1]           :=     160.0; // relative to rPosWait
GVL_XTS.StationParameter[nStationParameter].rReleaseDistance      :=     800.0; // relative to Mover.ActPos

nStationParameter := 60;
GVL_XTS.StationParameter[nStationParameter].eType                 := E_STATION_TYPE.STATION_PROCESS;
GVL_XTS.StationParameter[nStationParameter].sText                 := 'PRC_06_03';
GVL_XTS.StationParameter[nStationParameter].nConfiguredStopCount  :=       1;   // how many stops the mover has to make in this station

GVL_XTS.StationParameter[nStationParameter].rPosWait              :=    9500.0; // absolute modulo position
GVL_XTS.StationParameter[nStationParameter].rPosStop[1]           :=     240.0; // relative to rPosWait
GVL_XTS.StationParameter[nStationParameter].rReleaseDistance      :=     720.0; // relative to Mover.ActPos

nStationParameter := 61;
GVL_XTS.StationParameter[nStationParameter].eType                 := E_STATION_TYPE.STATION_PROCESS;
GVL_XTS.StationParameter[nStationParameter].sText                 := 'PRC_06_04';
GVL_XTS.StationParameter[nStationParameter].nConfiguredStopCount  :=       1;   // how many stops the mover has to make in this station

GVL_XTS.StationParameter[nStationParameter].rPosWait              :=    9500.0; // absolute modulo position
GVL_XTS.StationParameter[nStationParameter].rPosStop[1]           :=     320.0; // relative to rPosWait
GVL_XTS.StationParameter[nStationParameter].rReleaseDistance      :=     640.0; // relative to Mover.ActPos

nStationParameter := 62;
GVL_XTS.StationParameter[nStationParameter].eType                 := E_STATION_TYPE.STATION_PROCESS;
GVL_XTS.StationParameter[nStationParameter].sText                 := 'PRC_06_05';
GVL_XTS.StationParameter[nStationParameter].nConfiguredStopCount  :=       1;   // how many stops the mover has to make in this station

GVL_XTS.StationParameter[nStationParameter].rPosWait              :=    9500.0; // absolute modulo position
GVL_XTS.StationParameter[nStationParameter].rPosStop[1]           :=     400.0; // relative to rPosWait
GVL_XTS.StationParameter[nStationParameter].rReleaseDistance      :=     560.0; // relative to Mover.ActPos

nStationParameter := 63;
GVL_XTS.StationParameter[nStationParameter].eType                 := E_STATION_TYPE.STATION_PROCESS;
GVL_XTS.StationParameter[nStationParameter].sText                 := 'PRC_06_06';
GVL_XTS.StationParameter[nStationParameter].nConfiguredStopCount  :=       1;   // how many stops the mover has to make in this station

GVL_XTS.StationParameter[nStationParameter].rPosWait              :=    9500.0; // absolute modulo position
GVL_XTS.StationParameter[nStationParameter].rPosStop[1]           :=     480.0; // relative to rPosWait
GVL_XTS.StationParameter[nStationParameter].rReleaseDistance      :=     480.0; // relative to Mover.ActPos

nStationParameter := 64;
GVL_XTS.StationParameter[nStationParameter].eType                 := E_STATION_TYPE.STATION_PROCESS;
GVL_XTS.StationParameter[nStationParameter].sText                 := 'PRC_06_07';
GVL_XTS.StationParameter[nStationParameter].nConfiguredStopCount  :=       1;   // how many stops the mover has to make in this station

GVL_XTS.StationParameter[nStationParameter].rPosWait              :=    9500.0; // absolute modulo position
GVL_XTS.StationParameter[nStationParameter].rPosStop[1]           :=     560.0; // relative to rPosWait
GVL_XTS.StationParameter[nStationParameter].rReleaseDistance      :=     400.0; // relative to Mover.ActPos

nStationParameter := 65;
GVL_XTS.StationParameter[nStationParameter].eType                 := E_STATION_TYPE.STATION_PROCESS;
GVL_XTS.StationParameter[nStationParameter].sText                 := 'PRC_06_08';
GVL_XTS.StationParameter[nStationParameter].nConfiguredStopCount  :=       1;   // how many stops the mover has to make in this station

GVL_XTS.StationParameter[nStationParameter].rPosWait              :=    9500.0; // absolute modulo position
GVL_XTS.StationParameter[nStationParameter].rPosStop[1]           :=     640.0; // relative to rPosWait
GVL_XTS.StationParameter[nStationParameter].rReleaseDistance      :=     320.0; // relative to Mover.ActPos

nStationParameter := 66;
GVL_XTS.StationParameter[nStationParameter].eType                 := E_STATION_TYPE.STATION_PROCESS;
GVL_XTS.StationParameter[nStationParameter].sText                 := 'PRC_06_09';
GVL_XTS.StationParameter[nStationParameter].nConfiguredStopCount  :=       1;   // how many stops the mover has to make in this station

GVL_XTS.StationParameter[nStationParameter].rPosWait              :=    9500.0; // absolute modulo position
GVL_XTS.StationParameter[nStationParameter].rPosStop[1]           :=     720.0; // relative to rPosWait
GVL_XTS.StationParameter[nStationParameter].rReleaseDistance      :=     240.0; // relative to Mover.ActPos

nStationParameter := 67;
GVL_XTS.StationParameter[nStationParameter].eType                 := E_STATION_TYPE.STATION_PROCESS;
GVL_XTS.StationParameter[nStationParameter].sText                 := 'PRC_06_10';
GVL_XTS.StationParameter[nStationParameter].nConfiguredStopCount  :=       1;   // how many stops the mover has to make in this station

GVL_XTS.StationParameter[nStationParameter].rPosWait              :=    9500.0; // absolute modulo position
GVL_XTS.StationParameter[nStationParameter].rPosStop[1]           :=     800.0; // relative to rPosWait
GVL_XTS.StationParameter[nStationParameter].rReleaseDistance      :=     160.0; // relative to Mover.ActPos

nStationParameter := 68;
GVL_XTS.StationParameter[nStationParameter].eType                 := E_STATION_TYPE.STATION_PROCESS;
GVL_XTS.StationParameter[nStationParameter].sText                 := 'PRC_06_11';
GVL_XTS.StationParameter[nStationParameter].nConfiguredStopCount  :=       1;   // how many stops the mover has to make in this station

GVL_XTS.StationParameter[nStationParameter].rPosWait              :=    9500.0; // absolute modulo position
GVL_XTS.StationParameter[nStationParameter].rPosStop[1]           :=     880.0; // relative to rPosWait
GVL_XTS.StationParameter[nStationParameter].rReleaseDistance      :=      80.0; // relative to Mover.ActPos

nStationParameter := 69;
GVL_XTS.StationParameter[nStationParameter].eType                 := E_STATION_TYPE.STATION_PROCESS;
GVL_XTS.StationParameter[nStationParameter].sText                 := 'PRC_06_12';
GVL_XTS.StationParameter[nStationParameter].nConfiguredStopCount  :=       1;   // how many stops the mover has to make in this station

GVL_XTS.StationParameter[nStationParameter].rPosWait              :=    9500.0; // absolute modulo position
GVL_XTS.StationParameter[nStationParameter].rPosStop[1]           :=     960.0; // relative to rPosWait
GVL_XTS.StationParameter[nStationParameter].rReleaseDistance      :=      25.0; // relative to Mover.ActPos

//-----------------------------------------------------------------------------------------------------------------------------------------
// PRC 07 
//-----------------------------------------------------------------------------------------------------------------------------------------
nStationParameter := 70;
GVL_XTS.StationParameter[nStationParameter].eType                 := E_STATION_TYPE.STATION_PROCESS;
GVL_XTS.StationParameter[nStationParameter].sText                 := 'PRC_07_01';
GVL_XTS.StationParameter[nStationParameter].nConfiguredStopCount  :=       1;   // how many stops the mover has to make in this station

GVL_XTS.StationParameter[nStationParameter].rPosWait              :=   11500.0; // absolute modulo position
GVL_XTS.StationParameter[nStationParameter].rPosStop[1]           :=      80.0; // relative to rPosWait
GVL_XTS.StationParameter[nStationParameter].rReleaseDistance      :=     880.0; // relative to Mover.ActPos

nStationParameter := 71;
GVL_XTS.StationParameter[nStationParameter].eType                 := E_STATION_TYPE.STATION_PROCESS;
GVL_XTS.StationParameter[nStationParameter].sText                 := 'PRC_07_02';
GVL_XTS.StationParameter[nStationParameter].nConfiguredStopCount  :=       1;   // how many stops the mover has to make in this station

GVL_XTS.StationParameter[nStationParameter].rPosWait              :=   11500.0; // absolute modulo position
GVL_XTS.StationParameter[nStationParameter].rPosStop[1]           :=     160.0; // relative to rPosWait
GVL_XTS.StationParameter[nStationParameter].rReleaseDistance      :=     800.0; // relative to Mover.ActPos

nStationParameter := 72;
GVL_XTS.StationParameter[nStationParameter].eType                 := E_STATION_TYPE.STATION_PROCESS;
GVL_XTS.StationParameter[nStationParameter].sText                 := 'PRC_07_03';
GVL_XTS.StationParameter[nStationParameter].nConfiguredStopCount  :=       1;   // how many stops the mover has to make in this station

GVL_XTS.StationParameter[nStationParameter].rPosWait              :=   11500.0; // absolute modulo position
GVL_XTS.StationParameter[nStationParameter].rPosStop[1]           :=     240.0; // relative to rPosWait
GVL_XTS.StationParameter[nStationParameter].rReleaseDistance      :=     720.0; // relative to Mover.ActPos

nStationParameter := 73;
GVL_XTS.StationParameter[nStationParameter].eType                 := E_STATION_TYPE.STATION_PROCESS;
GVL_XTS.StationParameter[nStationParameter].sText                 := 'PRC_07_04';
GVL_XTS.StationParameter[nStationParameter].nConfiguredStopCount  :=       1;   // how many stops the mover has to make in this station

GVL_XTS.StationParameter[nStationParameter].rPosWait              :=   11500.0; // absolute modulo position
GVL_XTS.StationParameter[nStationParameter].rPosStop[1]           :=     320.0; // relative to rPosWait
GVL_XTS.StationParameter[nStationParameter].rReleaseDistance      :=     640.0; // relative to Mover.ActPos

nStationParameter := 74;
GVL_XTS.StationParameter[nStationParameter].eType                 := E_STATION_TYPE.STATION_PROCESS;
GVL_XTS.StationParameter[nStationParameter].sText                 := 'PRC_07_05';
GVL_XTS.StationParameter[nStationParameter].nConfiguredStopCount  :=       1;   // how many stops the mover has to make in this station

GVL_XTS.StationParameter[nStationParameter].rPosWait              :=   11500.0; // absolute modulo position
GVL_XTS.StationParameter[nStationParameter].rPosStop[1]           :=     400.0; // relative to rPosWait
GVL_XTS.StationParameter[nStationParameter].rReleaseDistance      :=     560.0; // relative to Mover.ActPos

nStationParameter := 75;
GVL_XTS.StationParameter[nStationParameter].eType                 := E_STATION_TYPE.STATION_PROCESS;
GVL_XTS.StationParameter[nStationParameter].sText                 := 'PRC_07_06';
GVL_XTS.StationParameter[nStationParameter].nConfiguredStopCount  :=       1;   // how many stops the mover has to make in this station

GVL_XTS.StationParameter[nStationParameter].rPosWait              :=   11500.0; // absolute modulo position
GVL_XTS.StationParameter[nStationParameter].rPosStop[1]           :=     480.0; // relative to rPosWait
GVL_XTS.StationParameter[nStationParameter].rReleaseDistance      :=     480.0; // relative to Mover.ActPos

nStationParameter := 76;
GVL_XTS.StationParameter[nStationParameter].eType                 := E_STATION_TYPE.STATION_PROCESS;
GVL_XTS.StationParameter[nStationParameter].sText                 := 'PRC_07_07';
GVL_XTS.StationParameter[nStationParameter].nConfiguredStopCount  :=       1;   // how many stops the mover has to make in this station

GVL_XTS.StationParameter[nStationParameter].rPosWait              :=   11500.0; // absolute modulo position
GVL_XTS.StationParameter[nStationParameter].rPosStop[1]           :=     560.0; // relative to rPosWait
GVL_XTS.StationParameter[nStationParameter].rReleaseDistance      :=     400.0; // relative to Mover.ActPos

nStationParameter := 77;
GVL_XTS.StationParameter[nStationParameter].eType                 := E_STATION_TYPE.STATION_PROCESS;
GVL_XTS.StationParameter[nStationParameter].sText                 := 'PRC_07_08';
GVL_XTS.StationParameter[nStationParameter].nConfiguredStopCount  :=       1;   // how many stops the mover has to make in this station

GVL_XTS.StationParameter[nStationParameter].rPosWait              :=   11500.0; // absolute modulo position
GVL_XTS.StationParameter[nStationParameter].rPosStop[1]           :=     640.0; // relative to rPosWait
GVL_XTS.StationParameter[nStationParameter].rReleaseDistance      :=     320.0; // relative to Mover.ActPos

nStationParameter := 78;
GVL_XTS.StationParameter[nStationParameter].eType                 := E_STATION_TYPE.STATION_PROCESS;
GVL_XTS.StationParameter[nStationParameter].sText                 := 'PRC_07_09';
GVL_XTS.StationParameter[nStationParameter].nConfiguredStopCount  :=       1;   // how many stops the mover has to make in this station

GVL_XTS.StationParameter[nStationParameter].rPosWait              :=   11500.0; // absolute modulo position
GVL_XTS.StationParameter[nStationParameter].rPosStop[1]           :=     720.0; // relative to rPosWait
GVL_XTS.StationParameter[nStationParameter].rReleaseDistance      :=     240.0; // relative to Mover.ActPos

nStationParameter := 79;
GVL_XTS.StationParameter[nStationParameter].eType                 := E_STATION_TYPE.STATION_PROCESS;
GVL_XTS.StationParameter[nStationParameter].sText                 := 'PRC_07_10';
GVL_XTS.StationParameter[nStationParameter].nConfiguredStopCount  :=       1;   // how many stops the mover has to make in this station

GVL_XTS.StationParameter[nStationParameter].rPosWait              :=   11500.0; // absolute modulo position
GVL_XTS.StationParameter[nStationParameter].rPosStop[1]           :=     800.0; // relative to rPosWait
GVL_XTS.StationParameter[nStationParameter].rReleaseDistance      :=     160.0; // relative to Mover.ActPos

nStationParameter := 80;
GVL_XTS.StationParameter[nStationParameter].eType                 := E_STATION_TYPE.STATION_PROCESS;
GVL_XTS.StationParameter[nStationParameter].sText                 := 'PRC_07_11';
GVL_XTS.StationParameter[nStationParameter].nConfiguredStopCount  :=       1;   // how many stops the mover has to make in this station

GVL_XTS.StationParameter[nStationParameter].rPosWait              :=   11500.0; // absolute modulo position
GVL_XTS.StationParameter[nStationParameter].rPosStop[1]           :=     880.0; // relative to rPosWait
GVL_XTS.StationParameter[nStationParameter].rReleaseDistance      :=      80.0; // relative to Mover.ActPos

nStationParameter := 81;
GVL_XTS.StationParameter[nStationParameter].eType                 := E_STATION_TYPE.STATION_PROCESS;
GVL_XTS.StationParameter[nStationParameter].sText                 := 'PRC_07_12';
GVL_XTS.StationParameter[nStationParameter].nConfiguredStopCount  :=       1;   // how many stops the mover has to make in this station

GVL_XTS.StationParameter[nStationParameter].rPosWait              :=   11500.0; // absolute modulo position
GVL_XTS.StationParameter[nStationParameter].rPosStop[1]           :=     960.0; // relative to rPosWait
GVL_XTS.StationParameter[nStationParameter].rReleaseDistance      :=      25.0; // relative to Mover.ActPos

//-----------------------------------------------------------------------------------------------------------------------------------------
// PRC 08 
//-----------------------------------------------------------------------------------------------------------------------------------------
nStationParameter := 82;
GVL_XTS.StationParameter[nStationParameter].eType                 := E_STATION_TYPE.STATION_PROCESS;
GVL_XTS.StationParameter[nStationParameter].sText                 := 'PRC_08_01';
GVL_XTS.StationParameter[nStationParameter].nConfiguredStopCount  :=       1;   // how many stops the mover has to make in this station

GVL_XTS.StationParameter[nStationParameter].rPosWait              :=   12750.0; // absolute modulo position
GVL_XTS.StationParameter[nStationParameter].rPosStop[1]           :=      80.0; // relative to rPosWait
GVL_XTS.StationParameter[nStationParameter].rReleaseDistance      :=     720.0; // relative to Mover.ActPos

nStationParameter := 83;
GVL_XTS.StationParameter[nStationParameter].eType                 := E_STATION_TYPE.STATION_PROCESS;
GVL_XTS.StationParameter[nStationParameter].sText                 := 'PRC_08_02';
GVL_XTS.StationParameter[nStationParameter].nConfiguredStopCount  :=       1;   // how many stops the mover has to make in this station

GVL_XTS.StationParameter[nStationParameter].rPosWait              :=   12750.0; // absolute modulo position
GVL_XTS.StationParameter[nStationParameter].rPosStop[1]           :=     160.0; // relative to rPosWait
GVL_XTS.StationParameter[nStationParameter].rReleaseDistance      :=     640.0; // relative to Mover.ActPos

nStationParameter := 84;
GVL_XTS.StationParameter[nStationParameter].eType                 := E_STATION_TYPE.STATION_PROCESS;
GVL_XTS.StationParameter[nStationParameter].sText                 := 'PRC_08_03';
GVL_XTS.StationParameter[nStationParameter].nConfiguredStopCount  :=       1;   // how many stops the mover has to make in this station

GVL_XTS.StationParameter[nStationParameter].rPosWait              :=   12750.0; // absolute modulo position
GVL_XTS.StationParameter[nStationParameter].rPosStop[1]           :=     240.0; // relative to rPosWait
GVL_XTS.StationParameter[nStationParameter].rReleaseDistance      :=     560.0; // relative to Mover.ActPos

nStationParameter := 85;
GVL_XTS.StationParameter[nStationParameter].eType                 := E_STATION_TYPE.STATION_PROCESS;
GVL_XTS.StationParameter[nStationParameter].sText                 := 'PRC_08_04';
GVL_XTS.StationParameter[nStationParameter].nConfiguredStopCount  :=       1;   // how many stops the mover has to make in this station

GVL_XTS.StationParameter[nStationParameter].rPosWait              :=   12750.0; // absolute modulo position
GVL_XTS.StationParameter[nStationParameter].rPosStop[1]           :=     320.0; // relative to rPosWait
GVL_XTS.StationParameter[nStationParameter].rReleaseDistance      :=     480.0; // relative to Mover.ActPos

nStationParameter := 86;
GVL_XTS.StationParameter[nStationParameter].eType                 := E_STATION_TYPE.STATION_PROCESS;
GVL_XTS.StationParameter[nStationParameter].sText                 := 'PRC_08_05';
GVL_XTS.StationParameter[nStationParameter].nConfiguredStopCount  :=       1;   // how many stops the mover has to make in this station

GVL_XTS.StationParameter[nStationParameter].rPosWait              :=   12750.0; // absolute modulo position
GVL_XTS.StationParameter[nStationParameter].rPosStop[1]           :=     400.0; // relative to rPosWait
GVL_XTS.StationParameter[nStationParameter].rReleaseDistance      :=     400.0; // relative to Mover.ActPos

nStationParameter := 87;
GVL_XTS.StationParameter[nStationParameter].eType                 := E_STATION_TYPE.STATION_PROCESS;
GVL_XTS.StationParameter[nStationParameter].sText                 := 'PRC_08_06';
GVL_XTS.StationParameter[nStationParameter].nConfiguredStopCount  :=       1;   // how many stops the mover has to make in this station

GVL_XTS.StationParameter[nStationParameter].rPosWait              :=   12750.0; // absolute modulo position
GVL_XTS.StationParameter[nStationParameter].rPosStop[1]           :=     480.0; // relative to rPosWait
GVL_XTS.StationParameter[nStationParameter].rReleaseDistance      :=     320.0; // relative to Mover.ActPos

nStationParameter := 88;
GVL_XTS.StationParameter[nStationParameter].eType                 := E_STATION_TYPE.STATION_PROCESS;
GVL_XTS.StationParameter[nStationParameter].sText                 := 'PRC_08_07';
GVL_XTS.StationParameter[nStationParameter].nConfiguredStopCount  :=       1;   // how many stops the mover has to make in this station

GVL_XTS.StationParameter[nStationParameter].rPosWait              :=   12750.0; // absolute modulo position
GVL_XTS.StationParameter[nStationParameter].rPosStop[1]           :=     560.0; // relative to rPosWait
GVL_XTS.StationParameter[nStationParameter].rReleaseDistance      :=     240.0; // relative to Mover.ActPos

nStationParameter := 89;
GVL_XTS.StationParameter[nStationParameter].eType                 := E_STATION_TYPE.STATION_PROCESS;
GVL_XTS.StationParameter[nStationParameter].sText                 := 'PRC_08_08';
GVL_XTS.StationParameter[nStationParameter].nConfiguredStopCount  :=       1;   // how many stops the mover has to make in this station

GVL_XTS.StationParameter[nStationParameter].rPosWait              :=   12750.0; // absolute modulo position
GVL_XTS.StationParameter[nStationParameter].rPosStop[1]           :=     640.0; // relative to rPosWait
GVL_XTS.StationParameter[nStationParameter].rReleaseDistance      :=     160.0; // relative to Mover.ActPos

nStationParameter := 90;
GVL_XTS.StationParameter[nStationParameter].eType                 := E_STATION_TYPE.STATION_PROCESS;
GVL_XTS.StationParameter[nStationParameter].sText                 := 'PRC_08_09';
GVL_XTS.StationParameter[nStationParameter].nConfiguredStopCount  :=       1;   // how many stops the mover has to make in this station

GVL_XTS.StationParameter[nStationParameter].rPosWait              :=   12750.0; // absolute modulo position
GVL_XTS.StationParameter[nStationParameter].rPosStop[1]           :=     720.0; // relative to rPosWait
GVL_XTS.StationParameter[nStationParameter].rReleaseDistance      :=      80.0; // relative to Mover.ActPos

nStationParameter := 91;
GVL_XTS.StationParameter[nStationParameter].eType                 := E_STATION_TYPE.STATION_PROCESS;
GVL_XTS.StationParameter[nStationParameter].sText                 := 'PRC_08_10';
GVL_XTS.StationParameter[nStationParameter].nConfiguredStopCount  :=       1;   // how many stops the mover has to make in this station

GVL_XTS.StationParameter[nStationParameter].rPosWait              :=   12750.0; // absolute modulo position
GVL_XTS.StationParameter[nStationParameter].rPosStop[1]           :=     800.0; // relative to rPosWait
GVL_XTS.StationParameter[nStationParameter].rReleaseDistance      :=      25.0; // relative to Mover.ActPos

//-----------------------------------------------------------------------------------------------------------------------------------------
// PRC 09 
//-----------------------------------------------------------------------------------------------------------------------------------------
nStationParameter := 92;
GVL_XTS.StationParameter[nStationParameter].eType                 := E_STATION_TYPE.STATION_PROCESS;
GVL_XTS.StationParameter[nStationParameter].sText                 := 'PRC_09_01';
GVL_XTS.StationParameter[nStationParameter].nConfiguredStopCount  :=       1;   // how many stops the mover has to make in this station

GVL_XTS.StationParameter[nStationParameter].rPosWait              :=   14500.0; // absolute modulo position
GVL_XTS.StationParameter[nStationParameter].rPosStop[1]           :=      80.0; // relative to rPosWait
GVL_XTS.StationParameter[nStationParameter].rReleaseDistance      :=     560.0; // relative to Mover.ActPos

nStationParameter := 93;
GVL_XTS.StationParameter[nStationParameter].eType                 := E_STATION_TYPE.STATION_PROCESS;
GVL_XTS.StationParameter[nStationParameter].sText                 := 'PRC_09_02';
GVL_XTS.StationParameter[nStationParameter].nConfiguredStopCount  :=       1;   // how many stops the mover has to make in this station

GVL_XTS.StationParameter[nStationParameter].rPosWait              :=   14500.0; // absolute modulo position
GVL_XTS.StationParameter[nStationParameter].rPosStop[1]           :=     160.0; // relative to rPosWait
GVL_XTS.StationParameter[nStationParameter].rReleaseDistance      :=     480.0; // relative to Mover.ActPos

nStationParameter := 94;
GVL_XTS.StationParameter[nStationParameter].eType                 := E_STATION_TYPE.STATION_PROCESS;
GVL_XTS.StationParameter[nStationParameter].sText                 := 'PRC_09_03';
GVL_XTS.StationParameter[nStationParameter].nConfiguredStopCount  :=       1;   // how many stops the mover has to make in this station

GVL_XTS.StationParameter[nStationParameter].rPosWait              :=   14500.0; // absolute modulo position
GVL_XTS.StationParameter[nStationParameter].rPosStop[1]           :=     240.0; // relative to rPosWait
GVL_XTS.StationParameter[nStationParameter].rReleaseDistance      :=     400.0; // relative to Mover.ActPos

nStationParameter := 95;
GVL_XTS.StationParameter[nStationParameter].eType                 := E_STATION_TYPE.STATION_PROCESS;
GVL_XTS.StationParameter[nStationParameter].sText                 := 'PRC_09_04';
GVL_XTS.StationParameter[nStationParameter].nConfiguredStopCount  :=       1;   // how many stops the mover has to make in this station

GVL_XTS.StationParameter[nStationParameter].rPosWait              :=   14500.0; // absolute modulo position
GVL_XTS.StationParameter[nStationParameter].rPosStop[1]           :=     320.0; // relative to rPosWait
GVL_XTS.StationParameter[nStationParameter].rReleaseDistance      :=     320.0; // relative to Mover.ActPos

nStationParameter := 96;
GVL_XTS.StationParameter[nStationParameter].eType                 := E_STATION_TYPE.STATION_PROCESS;
GVL_XTS.StationParameter[nStationParameter].sText                 := 'PRC_09_05';
GVL_XTS.StationParameter[nStationParameter].nConfiguredStopCount  :=       1;   // how many stops the mover has to make in this station

GVL_XTS.StationParameter[nStationParameter].rPosWait              :=   14500.0; // absolute modulo position
GVL_XTS.StationParameter[nStationParameter].rPosStop[1]           :=     400.0; // relative to rPosWait
GVL_XTS.StationParameter[nStationParameter].rReleaseDistance      :=     240.0; // relative to Mover.ActPos

nStationParameter := 97;
GVL_XTS.StationParameter[nStationParameter].eType                 := E_STATION_TYPE.STATION_PROCESS;
GVL_XTS.StationParameter[nStationParameter].sText                 := 'PRC_09_06';
GVL_XTS.StationParameter[nStationParameter].nConfiguredStopCount  :=       1;   // how many stops the mover has to make in this station

GVL_XTS.StationParameter[nStationParameter].rPosWait              :=   14500.0; // absolute modulo position
GVL_XTS.StationParameter[nStationParameter].rPosStop[1]           :=     480.0; // relative to rPosWait
GVL_XTS.StationParameter[nStationParameter].rReleaseDistance      :=     160.0; // relative to Mover.ActPos

nStationParameter := 98;
GVL_XTS.StationParameter[nStationParameter].eType                 := E_STATION_TYPE.STATION_PROCESS;
GVL_XTS.StationParameter[nStationParameter].sText                 := 'PRC_09_07';
GVL_XTS.StationParameter[nStationParameter].nConfiguredStopCount  :=       1;   // how many stops the mover has to make in this station

GVL_XTS.StationParameter[nStationParameter].rPosWait              :=   14500.0; // absolute modulo position
GVL_XTS.StationParameter[nStationParameter].rPosStop[1]           :=     560.0; // relative to rPosWait
GVL_XTS.StationParameter[nStationParameter].rReleaseDistance      :=      80.0; // relative to Mover.ActPos

nStationParameter := 99;
GVL_XTS.StationParameter[nStationParameter].eType                 := E_STATION_TYPE.STATION_PROCESS;
GVL_XTS.StationParameter[nStationParameter].sText                 := 'PRC_09_08';
GVL_XTS.StationParameter[nStationParameter].nConfiguredStopCount  :=       1;   // how many stops the mover has to make in this station

GVL_XTS.StationParameter[nStationParameter].rPosWait              :=   14500.0; // absolute modulo position
GVL_XTS.StationParameter[nStationParameter].rPosStop[1]           :=     640.0; // relative to rPosWait
GVL_XTS.StationParameter[nStationParameter].rReleaseDistance      :=      25.0; // relative to Mover.ActPos

//-----------------------------------------------------------------------------------------------------------------------------------------
// PRC 12 
//-----------------------------------------------------------------------------------------------------------------------------------------
nStationParameter := 110;
GVL_XTS.StationParameter[nStationParameter].eType                 := E_STATION_TYPE.STATION_PROCESS;
GVL_XTS.StationParameter[nStationParameter].sText                 := 'PRC_12_01';
GVL_XTS.StationParameter[nStationParameter].nConfiguredStopCount  :=       1;   // how many stops the mover has to make in this station

GVL_XTS.StationParameter[nStationParameter].rPosWait              :=   17000.0; // absolute modulo position
GVL_XTS.StationParameter[nStationParameter].rPosStop[1]           :=      80.0; // relative to rPosWait
GVL_XTS.StationParameter[nStationParameter].rReleaseDistance      :=     560.0; // relative to Mover.ActPos

nStationParameter := 111;
GVL_XTS.StationParameter[nStationParameter].eType                 := E_STATION_TYPE.STATION_PROCESS;
GVL_XTS.StationParameter[nStationParameter].sText                 := 'PRC_12_02';
GVL_XTS.StationParameter[nStationParameter].nConfiguredStopCount  :=       1;   // how many stops the mover has to make in this station

GVL_XTS.StationParameter[nStationParameter].rPosWait              :=   17000.0; // absolute modulo position
GVL_XTS.StationParameter[nStationParameter].rPosStop[1]           :=     160.0; // relative to rPosWait
GVL_XTS.StationParameter[nStationParameter].rReleaseDistance      :=     480.0; // relative to Mover.ActPos

nStationParameter := 112;
GVL_XTS.StationParameter[nStationParameter].eType                 := E_STATION_TYPE.STATION_PROCESS;
GVL_XTS.StationParameter[nStationParameter].sText                 := 'PRC_12_03';
GVL_XTS.StationParameter[nStationParameter].nConfiguredStopCount  :=       1;   // how many stops the mover has to make in this station

GVL_XTS.StationParameter[nStationParameter].rPosWait              :=   17000.0; // absolute modulo position
GVL_XTS.StationParameter[nStationParameter].rPosStop[1]           :=     240.0; // relative to rPosWait
GVL_XTS.StationParameter[nStationParameter].rReleaseDistance      :=     400.0; // relative to Mover.ActPos

nStationParameter := 113;
GVL_XTS.StationParameter[nStationParameter].eType                 := E_STATION_TYPE.STATION_PROCESS;
GVL_XTS.StationParameter[nStationParameter].sText                 := 'PRC_12_04';
GVL_XTS.StationParameter[nStationParameter].nConfiguredStopCount  :=       1;   // how many stops the mover has to make in this station

GVL_XTS.StationParameter[nStationParameter].rPosWait              :=   17000.0; // absolute modulo position
GVL_XTS.StationParameter[nStationParameter].rPosStop[1]           :=     320.0; // relative to rPosWait
GVL_XTS.StationParameter[nStationParameter].rReleaseDistance      :=     320.0; // relative to Mover.ActPos

nStationParameter := 114;
GVL_XTS.StationParameter[nStationParameter].eType                 := E_STATION_TYPE.STATION_PROCESS;
GVL_XTS.StationParameter[nStationParameter].sText                 := 'PRC_12_05';
GVL_XTS.StationParameter[nStationParameter].nConfiguredStopCount  :=       1;   // how many stops the mover has to make in this station

GVL_XTS.StationParameter[nStationParameter].rPosWait              :=   17000.0; // absolute modulo position
GVL_XTS.StationParameter[nStationParameter].rPosStop[1]           :=     400.0; // relative to rPosWait
GVL_XTS.StationParameter[nStationParameter].rReleaseDistance      :=     240.0; // relative to Mover.ActPos

nStationParameter := 115;
GVL_XTS.StationParameter[nStationParameter].eType                 := E_STATION_TYPE.STATION_PROCESS;
GVL_XTS.StationParameter[nStationParameter].sText                 := 'PRC_12_06';
GVL_XTS.StationParameter[nStationParameter].nConfiguredStopCount  :=       1;   // how many stops the mover has to make in this station

GVL_XTS.StationParameter[nStationParameter].rPosWait              :=   17000.0; // absolute modulo position
GVL_XTS.StationParameter[nStationParameter].rPosStop[1]           :=     480.0; // relative to rPosWait
GVL_XTS.StationParameter[nStationParameter].rReleaseDistance      :=     160.0; // relative to Mover.ActPos

nStationParameter := 116;
GVL_XTS.StationParameter[nStationParameter].eType                 := E_STATION_TYPE.STATION_PROCESS;
GVL_XTS.StationParameter[nStationParameter].sText                 := 'PRC_12_07';
GVL_XTS.StationParameter[nStationParameter].nConfiguredStopCount  :=       1;   // how many stops the mover has to make in this station

GVL_XTS.StationParameter[nStationParameter].rPosWait              :=   17000.0; // absolute modulo position
GVL_XTS.StationParameter[nStationParameter].rPosStop[1]           :=     560.0; // relative to rPosWait
GVL_XTS.StationParameter[nStationParameter].rReleaseDistance      :=      80.0; // relative to Mover.ActPos

nStationParameter := 117;
GVL_XTS.StationParameter[nStationParameter].eType                 := E_STATION_TYPE.STATION_PROCESS;
GVL_XTS.StationParameter[nStationParameter].sText                 := 'PRC_12_08';
GVL_XTS.StationParameter[nStationParameter].nConfiguredStopCount  :=       1;   // how many stops the mover has to make in this station

GVL_XTS.StationParameter[nStationParameter].rPosWait              :=   17000.0; // absolute modulo position
GVL_XTS.StationParameter[nStationParameter].rPosStop[1]           :=     640.0; // relative to rPosWait
GVL_XTS.StationParameter[nStationParameter].rReleaseDistance      :=      25.0; // relative to Mover.ActPos

//-----------------------------------------------------------------------------------------------------------------------------------------
//  PRC 13
//-----------------------------------------------------------------------------------------------------------------------------------------
nStationParameter := 118;
GVL_XTS.StationParameter[nStationParameter].eType                 := E_STATION_TYPE.STATION_PROCESS;
GVL_XTS.StationParameter[nStationParameter].sText                 := 'PRC_13';
GVL_XTS.StationParameter[nStationParameter].nConfiguredStopCount  :=      1;   // how many stops the mover has to make in this station

GVL_XTS.StationParameter[nStationParameter].rPosWait              :=  15500.0; // absolute modulo position
GVL_XTS.StationParameter[nStationParameter].rPosStop[1]           :=      0.0; // relative to rPosWait
GVL_XTS.StationParameter[nStationParameter].rReleaseDistance      :=     -5.0; // relative to Mover.ActPos

GVL_XTS.StationParameter[nStationParameter].rGap                  :=     78.0;
GVL_XTS.StationParameter[nStationParameter].rVelo                 :=   1500.0;

//-----------------------------------------------------------------------------------------------------------------------------------------
//  PRC 14
//-----------------------------------------------------------------------------------------------------------------------------------------
nStationParameter := 119;
GVL_XTS.StationParameter[nStationParameter].eType                 := E_STATION_TYPE.STATION_PROCESS;
GVL_XTS.StationParameter[nStationParameter].sText                 := 'PRC_14';
GVL_XTS.StationParameter[nStationParameter].nConfiguredStopCount  :=      1;   // how many stops the mover has to make in this station

GVL_XTS.StationParameter[nStationParameter].rPosWait              :=  16000.0; // absolute modulo position
GVL_XTS.StationParameter[nStationParameter].rPosStop[1]           :=      0.0; // relative to rPosWait
GVL_XTS.StationParameter[nStationParameter].rReleaseDistance      :=     -5.0; // relative to Mover.ActPos

//-----------------------------------------------------------------------------------------------------------------------------------------
// PRC 16 
//-----------------------------------------------------------------------------------------------------------------------------------------
nStationParameter := 134;
GVL_XTS.StationParameter[nStationParameter].eType                 := E_STATION_TYPE.STATION_PROCESS;
GVL_XTS.StationParameter[nStationParameter].sText                 := 'PRC_16_01';
GVL_XTS.StationParameter[nStationParameter].nConfiguredStopCount  :=       1;   // how many stops the mover has to make in this station

GVL_XTS.StationParameter[nStationParameter].rPosWait              :=   19500.0; // absolute modulo position
GVL_XTS.StationParameter[nStationParameter].rPosStop[1]           :=      80.0; // relative to rPosWait
GVL_XTS.StationParameter[nStationParameter].rReleaseDistance      :=    1040.0; // relative to Mover.ActPos

nStationParameter := 135;
GVL_XTS.StationParameter[nStationParameter].eType                 := E_STATION_TYPE.STATION_PROCESS;
GVL_XTS.StationParameter[nStationParameter].sText                 := 'PRC_16_02';
GVL_XTS.StationParameter[nStationParameter].nConfiguredStopCount  :=       1;   // how many stops the mover has to make in this station

GVL_XTS.StationParameter[nStationParameter].rPosWait              :=   19500.0; // absolute modulo position
GVL_XTS.StationParameter[nStationParameter].rPosStop[1]           :=     160.0; // relative to rPosWait
GVL_XTS.StationParameter[nStationParameter].rReleaseDistance      :=     960.0; // relative to Mover.ActPos

nStationParameter := 136;
GVL_XTS.StationParameter[nStationParameter].eType                 := E_STATION_TYPE.STATION_PROCESS;
GVL_XTS.StationParameter[nStationParameter].sText                 := 'PRC_16_03';
GVL_XTS.StationParameter[nStationParameter].nConfiguredStopCount  :=       1;   // how many stops the mover has to make in this station

GVL_XTS.StationParameter[nStationParameter].rPosWait              :=   19500.0; // absolute modulo position
GVL_XTS.StationParameter[nStationParameter].rPosStop[1]           :=     240.0; // relative to rPosWait
GVL_XTS.StationParameter[nStationParameter].rReleaseDistance      :=     880.0; // relative to Mover.ActPos

nStationParameter := 137;
GVL_XTS.StationParameter[nStationParameter].eType                 := E_STATION_TYPE.STATION_PROCESS;
GVL_XTS.StationParameter[nStationParameter].sText                 := 'PRC_16_04';
GVL_XTS.StationParameter[nStationParameter].nConfiguredStopCount  :=       1;   // how many stops the mover has to make in this station

GVL_XTS.StationParameter[nStationParameter].rPosWait              :=   19500.0; // absolute modulo position
GVL_XTS.StationParameter[nStationParameter].rPosStop[1]           :=     320.0; // relative to rPosWait
GVL_XTS.StationParameter[nStationParameter].rReleaseDistance      :=     800.0; // relative to Mover.ActPos

nStationParameter := 138;
GVL_XTS.StationParameter[nStationParameter].eType                 := E_STATION_TYPE.STATION_PROCESS;
GVL_XTS.StationParameter[nStationParameter].sText                 := 'PRC_16_05';
GVL_XTS.StationParameter[nStationParameter].nConfiguredStopCount  :=       1;   // how many stops the mover has to make in this station

GVL_XTS.StationParameter[nStationParameter].rPosWait              :=   19500.0; // absolute modulo position
GVL_XTS.StationParameter[nStationParameter].rPosStop[1]           :=     400.0; // relative to rPosWait
GVL_XTS.StationParameter[nStationParameter].rReleaseDistance      :=     720.0; // relative to Mover.ActPos

nStationParameter := 139;
GVL_XTS.StationParameter[nStationParameter].eType                 := E_STATION_TYPE.STATION_PROCESS;
GVL_XTS.StationParameter[nStationParameter].sText                 := 'PRC_16_06';
GVL_XTS.StationParameter[nStationParameter].nConfiguredStopCount  :=       1;   // how many stops the mover has to make in this station

GVL_XTS.StationParameter[nStationParameter].rPosWait              :=   19500.0; // absolute modulo position
GVL_XTS.StationParameter[nStationParameter].rPosStop[1]           :=     480.0; // relative to rPosWait
GVL_XTS.StationParameter[nStationParameter].rReleaseDistance      :=     640.0; // relative to Mover.ActPos

nStationParameter := 140;
GVL_XTS.StationParameter[nStationParameter].eType                 := E_STATION_TYPE.STATION_PROCESS;
GVL_XTS.StationParameter[nStationParameter].sText                 := 'PRC_16_07';
GVL_XTS.StationParameter[nStationParameter].nConfiguredStopCount  :=       1;   // how many stops the mover has to make in this station

